FUNCTION_BLOCK InputAts400MockStatusReady IMPLEMENTS IInputAts400

METHOD GetInputData : InputDataAts400
GetInputData.Ready := true;
END_METHOD

END_FUNCTION_BLOCK

(* stored: Version 1.1.0.1, ProductVersion 3.1.4024.12
   POU InputAts400MockStatusReady: Id {6a4def4d-68fb-4ef4-a204-f8db62137245}, SpecialFunc None
   Method GetInputData: Id {d2d647f8-c582-47dd-b0e4-dd103bdd8254} *)
